{attribute 'GeneratedUsingTerminal: EK1100-0000-0018'}
{attribute addProperty BoxType "EK1100-0000-0018"}
{attribute addProperty Id "Beckhoff_EM7xxxEK1122Beckhoff_EM7xxxEK1122_DEE9974A2A_0001_EM7004_0000_9995EM7004_866015E192A_0002_EM7004_0000_9996EM7004_7586CC95115A_0003_EM7004_0000_9997EM7004_7586CC95115A_0004_EM7004_0000_0016EM7004_5FA1DD22119A_0005_EM7004_0000_0017EM7004_0F97553F119A_0006_EM7004_0000_0018EM7004_0F97553F119"}
{attribute addProperty CRC "2537928878"}
{attribute addProperty Size "681"}
{attribute addProperty Name "Beckhoff EM7xxx"}
TYPE Beckhoff_EM7xxx_9745B8AE EXTENDS EK1100_1FC0878B :
STRUCT
	{attribute addProperty Name "Beckhoff EM7xxxEK1122"}
	{attribute addProperty PreviousPort "Beckhoff EM7xxx : B"}
	Beckhoff_EM7xxxEK1122 : Beckhoff_EM7xxxEK1122_DEE9974A;
	{attribute addProperty Name "A_0001(EM7004-0000-9995)"}
	{attribute addProperty PreviousPort "Beckhoff EM7xxxEK1122 : C"}
	A_0001_EM7004_0000_9995 : EM7004_866015E1;
	{attribute addProperty Name "A_0002(EM7004-0000-9996)"}
	{attribute addProperty PreviousPort "A_0001(EM7004-0000-9995) : B"}
	A_0002_EM7004_0000_9996 : EM7004_7586CC95;
	{attribute addProperty Name "A_0003(EM7004-0000-9997)"}
	{attribute addProperty PreviousPort "A_0002(EM7004-0000-9996) : B"}
	A_0003_EM7004_0000_9997 : EM7004_7586CC95;
	{attribute addProperty Name "A_0004(EM7004-0000-0016)"}
	{attribute addProperty PreviousPort "A_0003(EM7004-0000-9997) : B"}
	A_0004_EM7004_0000_0016 : EM7004_5FA1DD22;
	{attribute addProperty Name "A_0005(EM7004-0000-0017)"}
	{attribute addProperty PreviousPort "A_0004(EM7004-0000-0016) : B"}
	A_0005_EM7004_0000_0017 : EM7004_0F97553F;
	{attribute addProperty Name "A_0006(EM7004-0000-0018)"}
	{attribute addProperty PreviousPort "A_0005(EM7004-0000-0017) : B"}
	A_0006_EM7004_0000_0018 : EM7004_0F97553F;
END_STRUCT
END_TYPE

(* stored: Version 1.2.0.0, ProductVersion 3.1.4024.11
   DUT Beckhoff_EM7xxx_9745B8AE: Id {c490958a-c9cf-4841-9da5-630cbb84258f} *)
